/// calibration that is determined by calibration sequences of the unit (static offsets, shifts)
TYPE HandlingDataCalibration :
STRUCT
END_STRUCT
END_TYPE

(* stored: Version 1.1.0.1
   DUT HandlingDataCalibration: Id {d314c1cc-45f4-4ad2-9f55-69f1aff69b7d} *)
